FUNCTION_BLOCK ARRAY2VALUES_4_BYTE (* Service Interface Function Block Type *)
  (* Description: Copyright (c) 2014 Profactor GmbH This program and the accompanying materials are made available under the terms of the Eclipse Public License 2.0 which is available at https://www.eclipse.org/legal/epl-2.0/ SPDX-License-Identifier: EPL-2.0 *)
  (* Version 3.0, 2025-04-14, Patrick Aigner, changed package *)
  (* Version 1.0, 2014-07-09, Matthias Plasch, Profactor GmbH *)
  PACKAGE eclipse4diac::convert;
  {SET_ATTRIBUTE(eclipse4diac::core::GenericClassName, 'GEN_ARRAY2VALUES')}
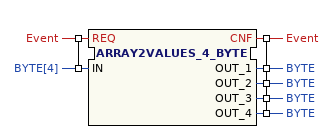
  EVENT_INPUT
    REQ WITH IN; (* Service Request *)
  END_EVENT
  EVENT_OUTPUT
    CNF WITH OUT_1, OUT_2, OUT_3, OUT_4; (* Confirmation of Requested Service *)
  END_EVENT
  VAR_INPUT
    IN : ARRAY [0..3] OF BYTE; (* Array input *)
  END_VAR
  VAR_OUTPUT
    OUT_1 : BYTE; (* output number 1 *)
    OUT_2 : BYTE; (* output number 2 *)
    OUT_3 : BYTE; (* output number 3 *)
    OUT_4 : BYTE; (* output number 4 *)
  END_VAR
END_FUNCTION_BLOCK
